(* Logix 5000 project; controller Transcat_L33ER vendor 1 type 14 code 107 rev 32.11; software revision 32.02; part 3 of 5 *)
(* tags used below, declared in another part *)
   AcsiiToReal1 : HexASCII_to_REAL;
   ActiveRecipe : Recipe;   // Active process recipe downloaded from the HMI recipe system and used by the PLC for automatic operation.
   AllDeviceEnable : BOOL;   // A bit to enable or disable the running of all devices
   AllReset : BOOL;   // Bit to reset Auto/Man, AutoRun, RecipeRun, TimedRunEnable to 0 from PLC
   alwaysOFF : BOOL;
   AnyAutoRun : BOOL;   // Bit that in on if ANY device is placed into Auto run (to signal pre-start beed)
   AnyAutoRunFlag : BOOL;   // A flag that indicates if any device is in Auto Run (used with pre-start beep logic)
   AnyManRunFlag : BOOL;   // A flag that indicates if any device is in Manual Run (used with pre-start beep logic)
   AnyManualRun : BOOL;   // Bit that in on if ANY device is placed into manual run (to signal pre-start beed)
   Auto_Run_All_Interlock : BOOL;   // Bit to interlock all devices running in Auto
   AutoActive : BOOL;   // Auto mode active
   AutoCampaignActive : BOOL;   // True after a new automatic campaign has started and remains true through interruptions until the campaign is completed o
   AutoRunRequest : BOOL;   // True when the automatic state machine is in RUNNING and automatic device operation is requested.
   AutoStartOS : BOOL;   // Auto Start One-Shot
   AutoState : DINT;   // Current automatic process state. 0=IDLE, 10=ARMED, 20=RUNNING, 30=INTERLOCKED
   AutoStopOS : BOOL;   // Auto Stop One-Shot
   Beep : BOOL;   // Bit to Activte Beacon Alarm
   bronkhorstReal : REAL[50];   // data from Bonkhorst - convertred to real values
   BronkOutArr : DINT[3];   // 3 Outputs from Flow controllers 0 - 100% = 0 - 32000
   BronkRealInArr : REAL[100];
   ConversionError : BOOL;
   ConvertedFloat : REAL;
   CV_101_Output : ALIAS FOR TC_Remote_IO:5:O.1;   // CV_101 - 3 Way Valve - Recyle / Process
   dataIndex : DINT;   // Bronkhorst Data Index
   Device : Device[20];
   dNum : DINT;   // The index of the current device being processed
   EstopActive : BOOL;   // E
   EstopFalutResetTOF : TIMER;   // Timer to hold reset bit to allow all drives to reset
   EStopResetPulse : BOOL;   // One-scan pulse used to clear all 14 E-stop interlocks - allows reset of estop interlocks from physical reset button on V
   EStopResetRequired : BOOL;   // Indicates that an estop was actived and it's awaiting reset
   FT103 : BronkhorstFlowMeter;
   FT104 : BronkhorstFlowMeter;
   FT105 : BronkhorstFlowMeter;
   HMI_AllReset : BOOL;   // Bit to reset Auto/Man, AutoRun, RecipeRun, TimedRunEnable to 0 from HMI
   HMI_AutoStart : BOOL;   // Starts all devices in AUTO
   HMI_AutoStop : BOOL;   // Stops all devices in AUTO
   HMI_ProcessReset : BOOL;   // Bit to clear the process hold/inteerlock when all other device interlocks are cleared
   HMI_RecipeStart : BOOL;   // Bit to start and stop recipe from HMI
   NewAutoCampaign : BOOL;   // One-scan pulse generated when the operator starts a new automatic campaign; used to initialize campaign-specific device
   NewDataToggle : BOOL;
   RecipeStart : BOOL;   // Bit to start and stop a recipe execution from PLC logic
   resultIndex : DINT;   // Bronkhorst Real Result Index
   StartBeepTimer : TIMER;   // Timer to sound the beep alarm before starting a device
   TempHexIn : SINT[8];   // Place to copy 8 SINT for proessing by AOI
   TestBit1 : BOOL;   // Just a test bit - does not do anything
(* MainProgram, continued *)

ROUTINE _13_CV101_3_Way_Dosing_Value   (* ladder *)
// 3 way valve to switch between recyle and feed to process
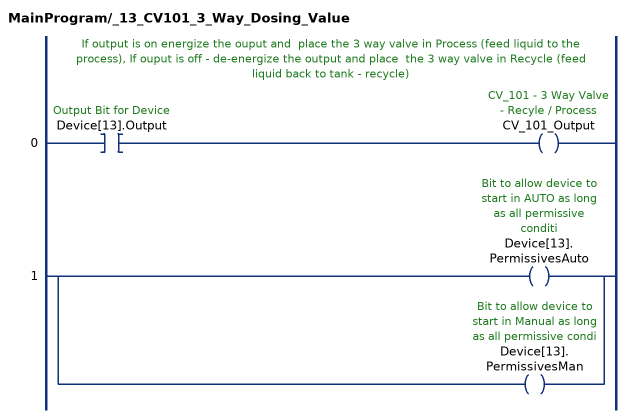
   // If output is on energize the ouput and  place the 3 way valve in Process (feed liquid to the process), If ouput is off - de-energize the output and place  the 3 way valve in Recycle (feed liquid back to tank - recycle)
   0: XIC(Device[13].Output)OTE(CV_101_Output);
   1: [OTE(Device[13].PermissivesAuto) ,OTE(Device[13].PermissivesMan) ];
END_ROUTINE

ROUTINE AutoControl   (* ladder *)
// Place where Auto device control logic lives
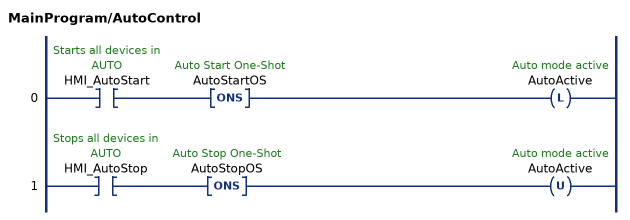
   0: XIC(HMI_AutoStart)ONS(AutoStartOS)OTL(AutoActive);
   1: XIC(HMI_AutoStop)ONS(AutoStopOS)OTU(AutoActive);
END_ROUTINE

ROUTINE AutoStateMachine   (* ladder *)
// Logic to Run system in Auto using a state machine
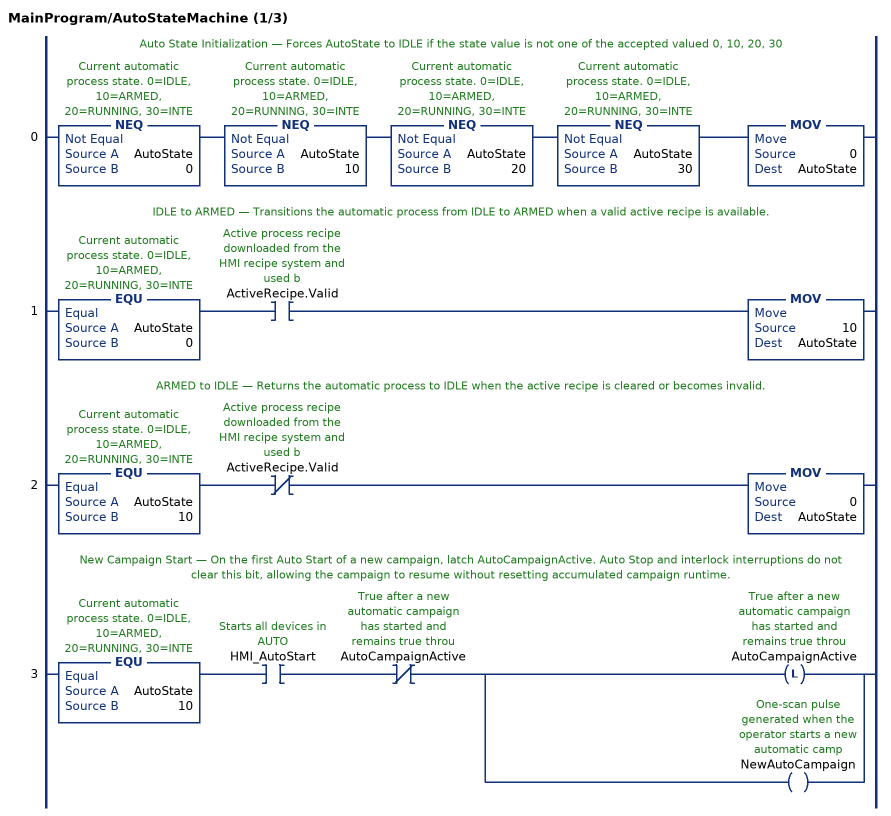
   // Auto State Initialization — Forces AutoState to IDLE if the state value is not one of the accepted valued 0, 10, 20, 30
   0: NEQ(AutoState,0)NEQ(AutoState,10)NEQ(AutoState,20)NEQ(AutoState,30)MOV(0,AutoState);
   // IDLE to ARMED — Transitions the automatic process from IDLE to ARMED when a valid active recipe is available.
   1: EQU(AutoState,0)XIC(ActiveRecipe.Valid)MOV(10,AutoState);
   // ARMED to IDLE — Returns the automatic process to IDLE when the active recipe is cleared or becomes invalid.
   2: EQU(AutoState,10)XIO(ActiveRecipe.Valid)MOV(0,AutoState);
   // New Campaign Start — On the first Auto Start of a new campaign, latch AutoCampaignActive. Auto Stop and interlock interruptions do not clear this bit, allowing the campaign to resume without resetting accumulated campaign runtime.
   3: EQU(AutoState,10)XIC(HMI_AutoStart)XIO(AutoCampaignActive)[OTL(AutoCampaignActive) ,OTE(NewAutoCampaign) ];
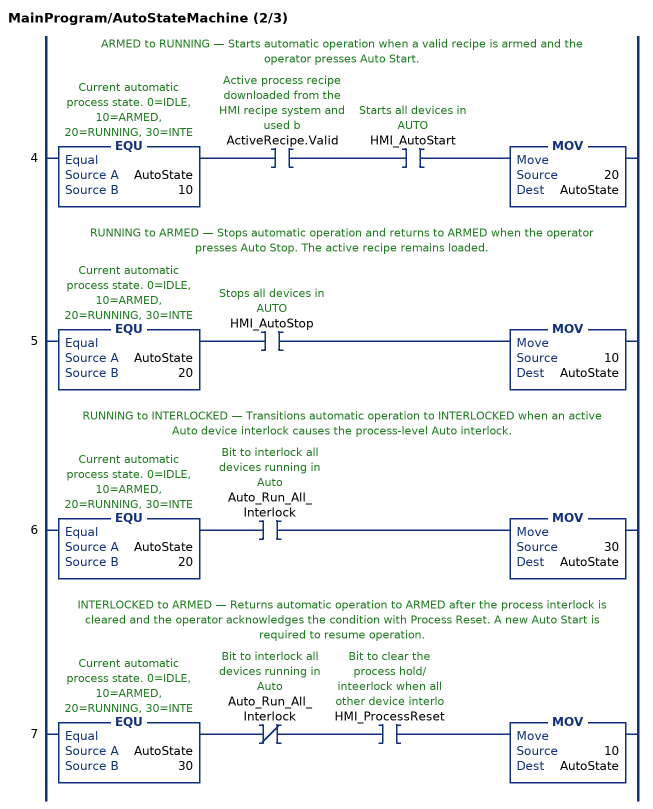
   // ARMED to RUNNING — Starts automatic operation when a valid recipe is armed and the operator presses Auto Start.
   4: EQU(AutoState,10)XIC(ActiveRecipe.Valid)XIC(HMI_AutoStart)MOV(20,AutoState);
   // RUNNING to ARMED — Stops automatic operation and returns to ARMED when the operator presses Auto Stop. The active recipe remains loaded.
   5: EQU(AutoState,20)XIC(HMI_AutoStop)MOV(10,AutoState);
   // RUNNING to INTERLOCKED — Transitions automatic operation to INTERLOCKED when an active Auto device interlock causes the process-level Auto interlock.
   6: EQU(AutoState,20)XIC(Auto_Run_All_Interlock)MOV(30,AutoState);
   // INTERLOCKED to ARMED — Returns automatic operation to ARMED after the process interlock is cleared and the operator acknowledges the condition with Process Reset. A new Auto Start is required to resume operation.
   7: EQU(AutoState,30)XIO(Auto_Run_All_Interlock)XIC(HMI_ProcessReset)MOV(10,AutoState);
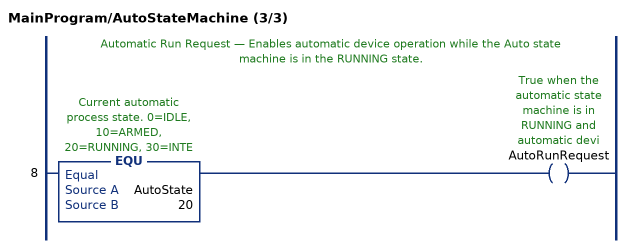
   // Automatic Run Request — Enables automatic device operation while the Auto state machine is in the RUNNING state.
   8: EQU(AutoState,20)OTE(AutoRunRequest);
END_ROUTINE

ROUTINE BronkDataMapping   (* structured text *)
// Map FT UDT elements to data to/from Bronkhorst Anybus Gateway
   FT103.AlarmID := Anybus_ETH_SER:I.Data[200];
   FT104.AlarmID := Anybus_ETH_SER:I.Data[201];
   FT105.AlarmID := Anybus_ETH_SER:I.Data[202];
   
   FT103.PV_R := BronkRealInArr[0];
   FT103.TempC := BronkRealInArr[1];
   FT103.Density := BronkRealInArr[2];
   FT103.SP_R := BronkRealInArr[3];
   FT103.Totalizer := BronkRealInArr[4];
   
   FT104.PV_R := BronkRealInArr[5];
   FT104.TempC := BronkRealInArr[6];
   FT104.Density := BronkRealInArr[7];
   FT104.SP_R := BronkRealInArr[8];
   FT104.Totalizer := BronkRealInArr[9];
   
   FT105.PV_R := BronkRealInArr[10];
   FT105.TempC := BronkRealInArr[11];
   FT105.Density := BronkRealInArr[12];
   FT105.SP_R := BronkRealInArr[13];
   FT105.Totalizer := BronkRealInArr[14];
   
   FT103.OT_R := (BronkOutArr[0]) / 167681.5;
   FT104.OT_R := (BronkOutArr[1]) / 167681.5;
   FT105.OT_R := (BronkOutArr[2]) / 167681.5;
END_ROUTINE

ROUTINE Bronkhorst_Data   (* ladder *)
// read and write data to/from the EIP instance and convert to/from 8 byte to/from floating point
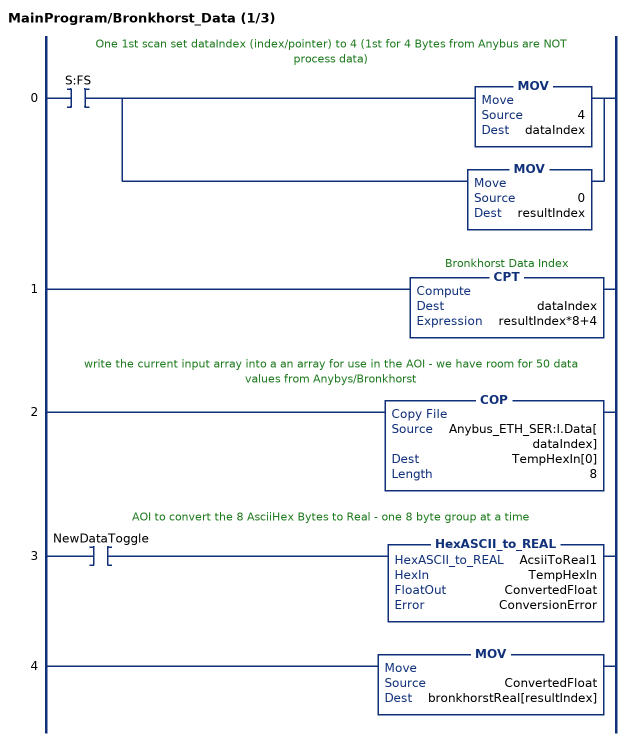
   // One 1st scan set dataIndex (index/pointer) to 4 (1st for 4 Bytes from Anybus are NOT process data)
   0: XIC(S:FS)[MOV(4,dataIndex) ,MOV(0,resultIndex) ];
   1: CPT(dataIndex,resultIndex*8+4);
   // write the current input array into a an array for use in the AOI - we have room for 50 data values from Anybys/Bronkhorst
   2: COP(Anybus_ETH_SER:I.Data[dataIndex],TempHexIn[0],8);
   // AOI to convert the 8 AsciiHex Bytes to Real - one 8 byte group at a time
   3: XIC(NewDataToggle)HexASCII_to_REAL(AcsiiToReal1,TempHexIn,ConvertedFloat,ConversionError);
   4: MOV(ConvertedFloat,bronkhorstReal[resultIndex]);
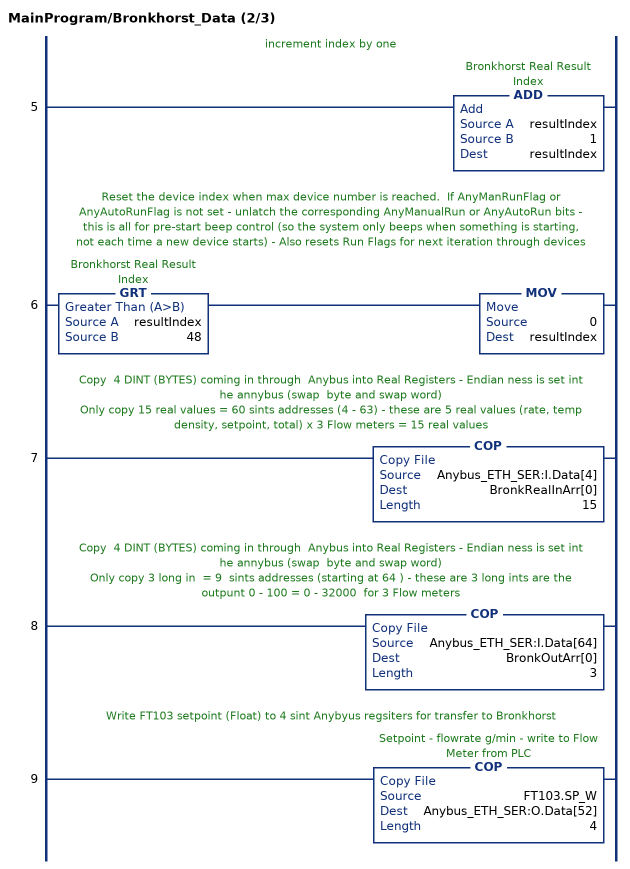
   // increment index by one
   5: ADD(resultIndex,1,resultIndex);
   // Reset the device index when max device number is reached.  If AnyManRunFlag or AnyAutoRunFlag is not set - unlatch the corresponding AnyManualRun or AnyAutoRun bits - this is all for pre-start beep control (so the system only beeps when something is starting, not each time a new device starts) - Also resets Run Flags for next iteration through devices
   6: GRT(resultIndex,48)MOV(0,resultIndex);
   // Copy  4 DINT (BYTES) coming in through  Anybus into Real Registers - Endian ness is set int he annybus (swap  byte and swap word)
   // Only copy 15 real values = 60 sints addresses (4 - 63) - these are 5 real values (rate, temp density, setpoint, total) x 3 Flow meters = 15 real values
   7: COP(Anybus_ETH_SER:I.Data[4],BronkRealInArr[0],15);
   // Copy  4 DINT (BYTES) coming in through  Anybus into Real Registers - Endian ness is set int he annybus (swap  byte and swap word)
   // Only copy 3 long in  = 9  sints addresses (starting at 64 ) - these are 3 long ints are the outpunt 0 - 100 = 0 - 32000  for 3 Flow meters
   8: COP(Anybus_ETH_SER:I.Data[64],BronkOutArr[0],3);
   // Write FT103 setpoint (Float) to 4 sint Anybyus regsiters for transfer to Bronkhorst
   9: COP(FT103.SP_W,Anybus_ETH_SER:O.Data[52],4);
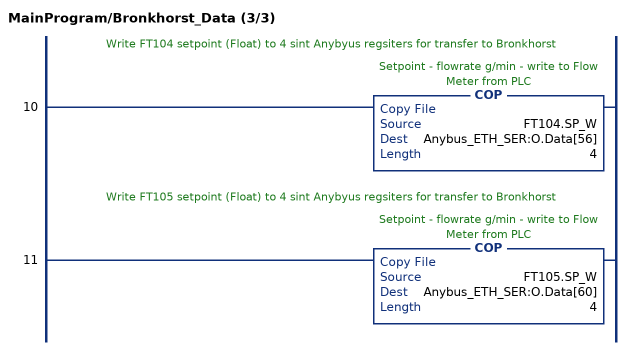
   // Write FT104 setpoint (Float) to 4 sint Anybyus regsiters for transfer to Bronkhorst
   10: COP(FT104.SP_W,Anybus_ETH_SER:O.Data[56],4);
   // Write FT105 setpoint (Float) to 4 sint Anybyus regsiters for transfer to Bronkhorst
   11: COP(FT105.SP_W,Anybus_ETH_SER:O.Data[60],4);
END_ROUTINE

ROUTINE DeviceLogic   (* ladder *)
// Process the logic for each device with index and indirect addressing.
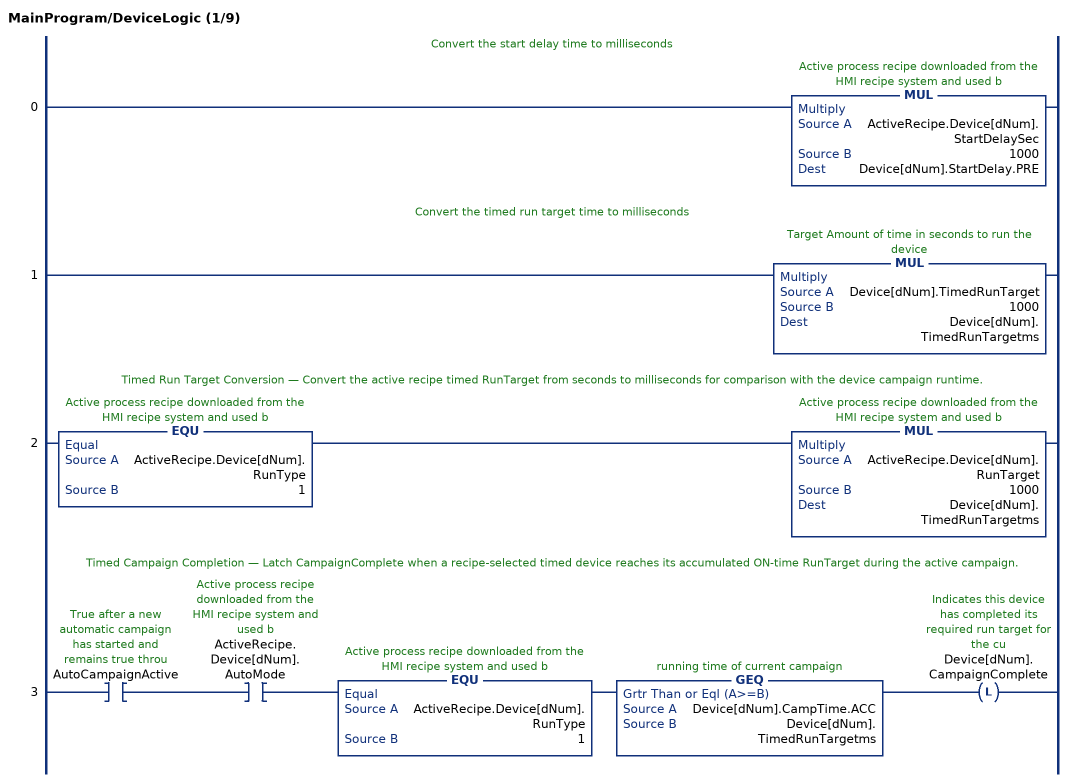
   // Convert the start delay time to milliseconds
   0: MUL(ActiveRecipe.Device[dNum].StartDelaySec,1000,Device[dNum].StartDelay.PRE);
   // Convert the timed run target time to milliseconds
   1: MUL(Device[dNum].TimedRunTarget,1000,Device[dNum].TimedRunTargetms);
   // Timed Run Target Conversion — Convert the active recipe timed RunTarget from seconds to milliseconds for comparison with the device campaign runtime.
   2: EQU(ActiveRecipe.Device[dNum].RunType,1)MUL(ActiveRecipe.Device[dNum].RunTarget,1000,Device[dNum].TimedRunTargetms);
   // Timed Campaign Completion — Latch CampaignComplete when a recipe-selected timed device reaches its accumulated ON-time RunTarget during the active campaign.
   3: XIC(AutoCampaignActive)XIC(ActiveRecipe.Device[dNum].AutoMode)EQU(ActiveRecipe.Device[dNum].RunType,1)GEQ(Device[dNum].CampTime.ACC,Device[dNum].TimedRunTargetms)OTL(Device[dNum].CampaignComplete);
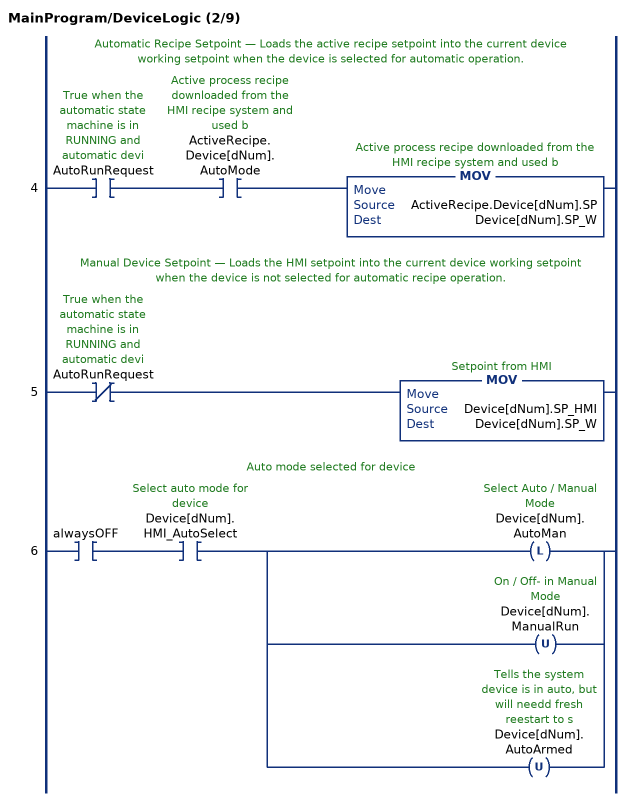
   // Automatic Recipe Setpoint — Loads the active recipe setpoint into the current device working setpoint when the device is selected for automatic operation.
   4: XIC(AutoRunRequest)XIC(ActiveRecipe.Device[dNum].AutoMode)MOV(ActiveRecipe.Device[dNum].SP,Device[dNum].SP_W);
   // Manual Device Setpoint — Loads the HMI setpoint into the current device working setpoint when the device is not selected for automatic recipe operation.
   5: XIO(AutoRunRequest)MOV(Device[dNum].SP_HMI,Device[dNum].SP_W);
   // Auto mode selected for device
   6: XIC(alwaysOFF)XIC(Device[dNum].HMI_AutoSelect)[OTL(Device[dNum].AutoMan) ,OTU(Device[dNum].ManualRun) ,OTU(Device[dNum].AutoArmed) ];
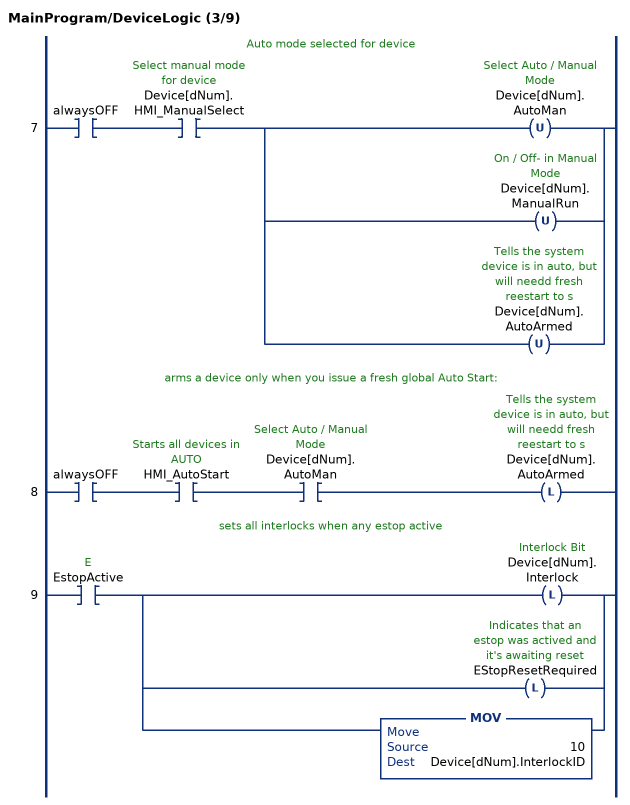
   // Auto mode selected for device
   7: XIC(alwaysOFF)XIC(Device[dNum].HMI_ManualSelect)[OTU(Device[dNum].AutoMan) ,[OTU(Device[dNum].ManualRun) ,OTU(Device[dNum].AutoArmed) ] ];
   // arms a device only when you issue a fresh global Auto Start:
   8: XIC(alwaysOFF)XIC(HMI_AutoStart)XIC(Device[dNum].AutoMan)OTL(Device[dNum].AutoArmed);
   // sets all interlocks when any estop active
   9: XIC(EstopActive)[OTL(Device[dNum].Interlock) ,OTL(EStopResetRequired) ,MOV(10,Device[dNum].InterlockID) ];
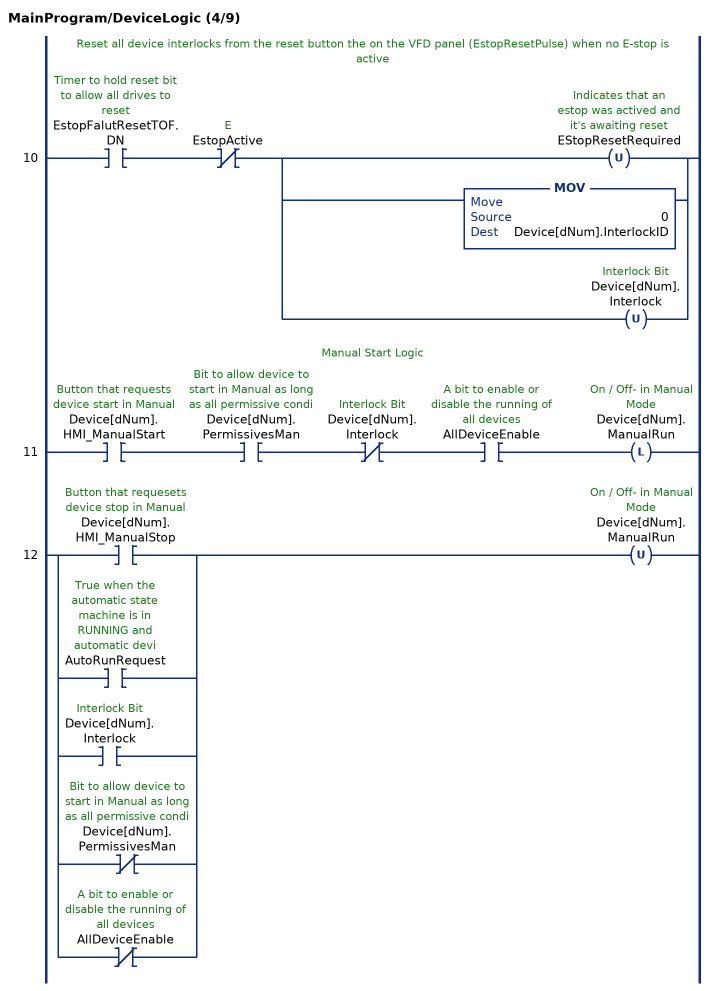
   // Reset all device interlocks from the reset button the on the VFD panel (EstopResetPulse) when no E-stop is active
   10: XIC(EstopFalutResetTOF.DN)XIO(EstopActive)[OTU(EStopResetRequired) ,MOV(0,Device[dNum].InterlockID) ,OTU(Device[dNum].Interlock) ];
   // Manual Start Logic
   11: XIC(Device[dNum].HMI_ManualStart)XIC(Device[dNum].PermissivesMan)XIO(Device[dNum].Interlock)XIC(AllDeviceEnable)OTL(Device[dNum].ManualRun);
   12: [XIC(Device[dNum].HMI_ManualStop) ,XIC(AutoRunRequest) ,XIC(Device[dNum].Interlock) ,XIO(Device[dNum].PermissivesMan) ,XIO(AllDeviceEnable) ]OTU(Device[dNum].ManualRun);
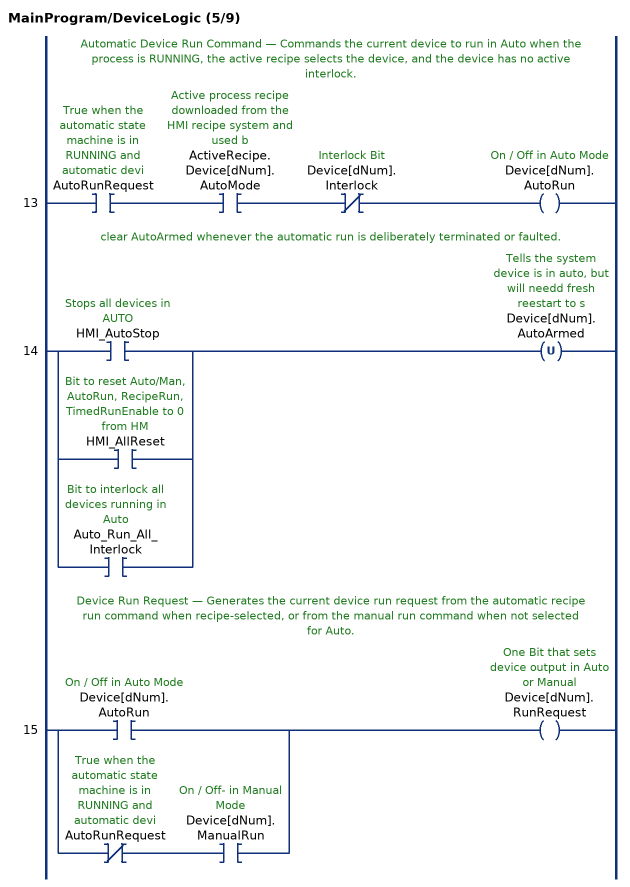
   // Automatic Device Run Command — Commands the current device to run in Auto when the process is RUNNING, the active recipe selects the device, and the device has no active interlock.
   13: XIC(AutoRunRequest)XIC(ActiveRecipe.Device[dNum].AutoMode)XIO(Device[dNum].Interlock)OTE(Device[dNum].AutoRun);
   // clear AutoArmed whenever the automatic run is deliberately terminated or faulted.
   14: [XIC(HMI_AutoStop) ,[XIC(HMI_AllReset) ,XIC(Auto_Run_All_Interlock) ] ]OTU(Device[dNum].AutoArmed);
   // Device Run Request — Generates the current device run request from the automatic recipe run command when recipe-selected, or from the manual run command when not selected for Auto.
   15: [XIC(Device[dNum].AutoRun) ,XIO(AutoRunRequest) XIC(Device[dNum].ManualRun) ]OTE(Device[dNum].RunRequest);
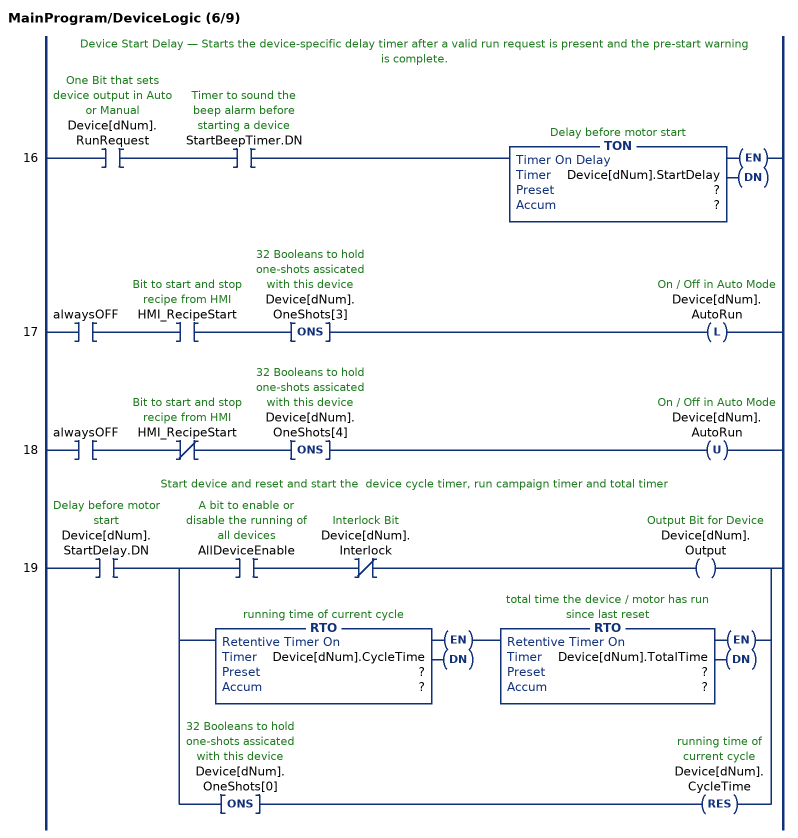
   // Device Start Delay — Starts the device-specific delay timer after a valid run request is present and the pre-start warning is complete.
   16: XIC(Device[dNum].RunRequest)XIC(StartBeepTimer.DN)TON(Device[dNum].StartDelay,?,?);
   17: XIC(alwaysOFF)XIC(HMI_RecipeStart)ONS(Device[dNum].OneShots[3])OTL(Device[dNum].AutoRun);
   18: XIC(alwaysOFF)XIO(HMI_RecipeStart)ONS(Device[dNum].OneShots[4])OTU(Device[dNum].AutoRun);
   // Start device and reset and start the  device cycle timer, run campaign timer and total timer
   19: XIC(Device[dNum].StartDelay.DN)[XIC(AllDeviceEnable) XIO(Device[dNum].Interlock) OTE(Device[dNum].Output) ,[RTO(Device[dNum].CycleTime,?,?) RTO(Device[dNum].TotalTime,?,?) ,ONS(Device[dNum].OneShots[0]) RES(Device[dNum].CycleTime) ] ];
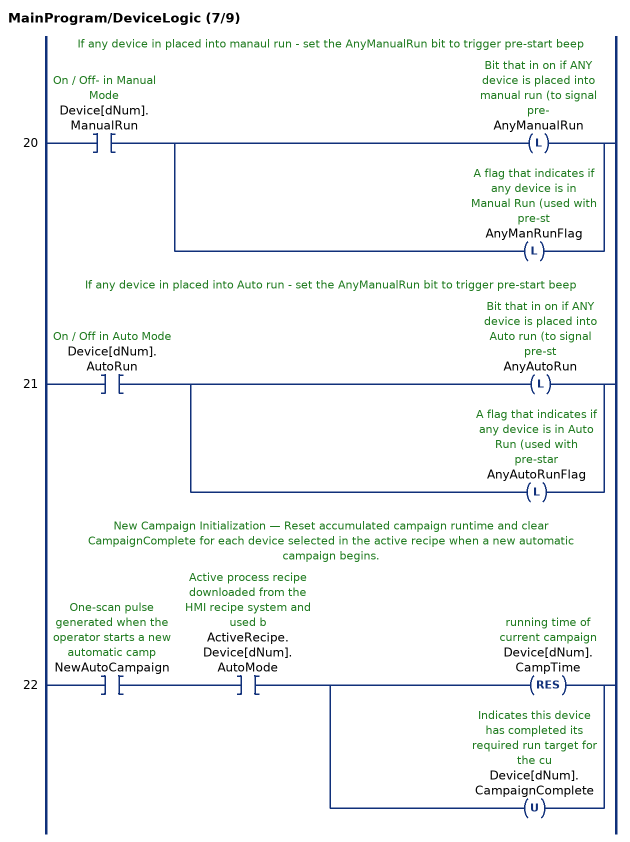
   // If any device in placed into manaul run - set the AnyManualRun bit to trigger pre-start beep
   20: XIC(Device[dNum].ManualRun)[OTL(AnyManualRun) ,OTL(AnyManRunFlag) ];
   // If any device in placed into Auto run - set the AnyManualRun bit to trigger pre-start beep
   21: XIC(Device[dNum].AutoRun)[OTL(AnyAutoRun) ,OTL(AnyAutoRunFlag) ];
   // New Campaign Initialization — Reset accumulated campaign runtime and clear CampaignComplete for each device selected in the active recipe when a new automatic campaign begins.
   22: XIC(NewAutoCampaign)XIC(ActiveRecipe.Device[dNum].AutoMode)[RES(Device[dNum].CampTime) ,OTU(Device[dNum].CampaignComplete) ];
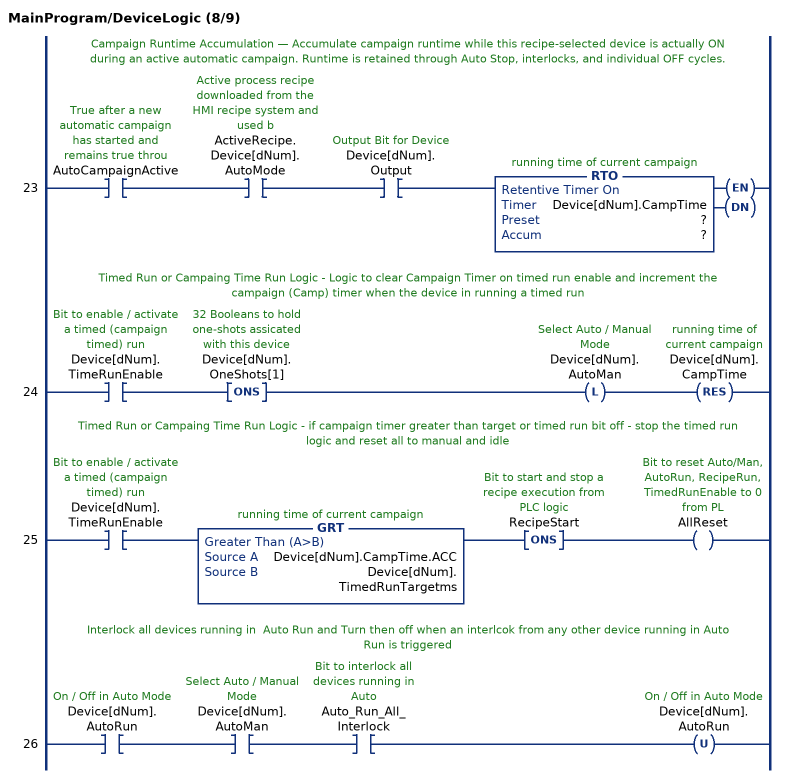
   // Campaign Runtime Accumulation — Accumulate campaign runtime while this recipe-selected device is actually ON during an active automatic campaign. Runtime is retained through Auto Stop, interlocks, and individual OFF cycles.
   23: XIC(AutoCampaignActive)XIC(ActiveRecipe.Device[dNum].AutoMode)XIC(Device[dNum].Output)RTO(Device[dNum].CampTime,?,?);
   // Timed Run or Campaing Time Run Logic - Logic to clear Campaign Timer on timed run enable and increment the campaign (Camp) timer when the device in running a timed run
   24: XIC(Device[dNum].TimeRunEnable)ONS(Device[dNum].OneShots[1])OTL(Device[dNum].AutoMan)RES(Device[dNum].CampTime);
   // Timed Run or Campaing Time Run Logic - if campaign timer greater than target or timed run bit off - stop the timed run logic and reset all to manual and idle
   25: XIC(Device[dNum].TimeRunEnable)GRT(Device[dNum].CampTime.ACC,Device[dNum].TimedRunTargetms)ONS(RecipeStart)OTE(AllReset);
   // Interlock all devices running in  Auto Run and Turn then off when an interlcok from any other device running in Auto Run is triggered
   26: XIC(Device[dNum].AutoRun)XIC(Device[dNum].AutoMan)XIC(Auto_Run_All_Interlock)OTU(Device[dNum].AutoRun);
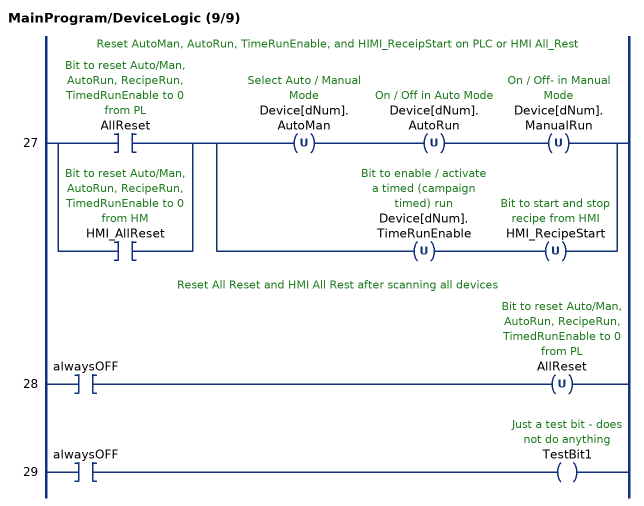
   // Reset AutoMan, AutoRun, TimeRunEnable, and HIMI_ReceipStart on PLC or HMI All_Rest
   27: [XIC(AllReset) ,XIC(HMI_AllReset) ][OTU(Device[dNum].AutoMan) OTU(Device[dNum].AutoRun) OTU(Device[dNum].ManualRun) ,OTU(Device[dNum].TimeRunEnable) OTU(HMI_RecipeStart) ];
   // Reset All Reset and HMI All Rest after scanning all devices
   28: XIC(alwaysOFF)OTU(AllReset);
   29: XIC(alwaysOFF)OTE(TestBit1);
END_ROUTINE

ROUTINE DeviceManager   (* ladder *)
// Loop through all devices each scan
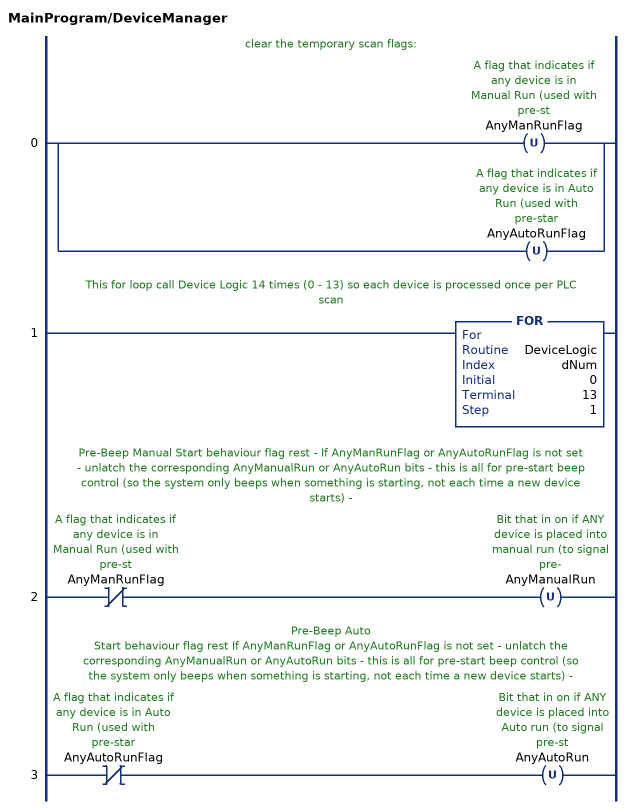
   // clear the temporary scan flags:
   0: [OTU(AnyManRunFlag) ,OTU(AnyAutoRunFlag) ];
   // This for loop call Device Logic 14 times (0 - 13) so each device is processed once per PLC scan
   1: FOR(DeviceLogic,dNum,0,13,1);
   // Pre-Beep Manual Start behaviour flag rest - If AnyManRunFlag or AnyAutoRunFlag is not set - unlatch the corresponding AnyManualRun or AnyAutoRun bits - this is all for pre-start beep control (so the system only beeps when something is starting, not each time a new device starts) -
   2: XIO(AnyManRunFlag)OTU(AnyManualRun);
   // Pre-Beep Auto
   //  Start behaviour flag rest If AnyManRunFlag or AnyAutoRunFlag is not set - unlatch the corresponding AnyManualRun or AnyAutoRun bits - this is all for pre-start beep control (so the system only beeps when something is starting, not each time a new device starts) -
   3: XIO(AnyAutoRunFlag)OTU(AnyAutoRun);
END_ROUTINE
